// Mitsubishi GX Works2 project: 0206 MPS회로   PLC: Q03UDV

PROGRAM MAIN
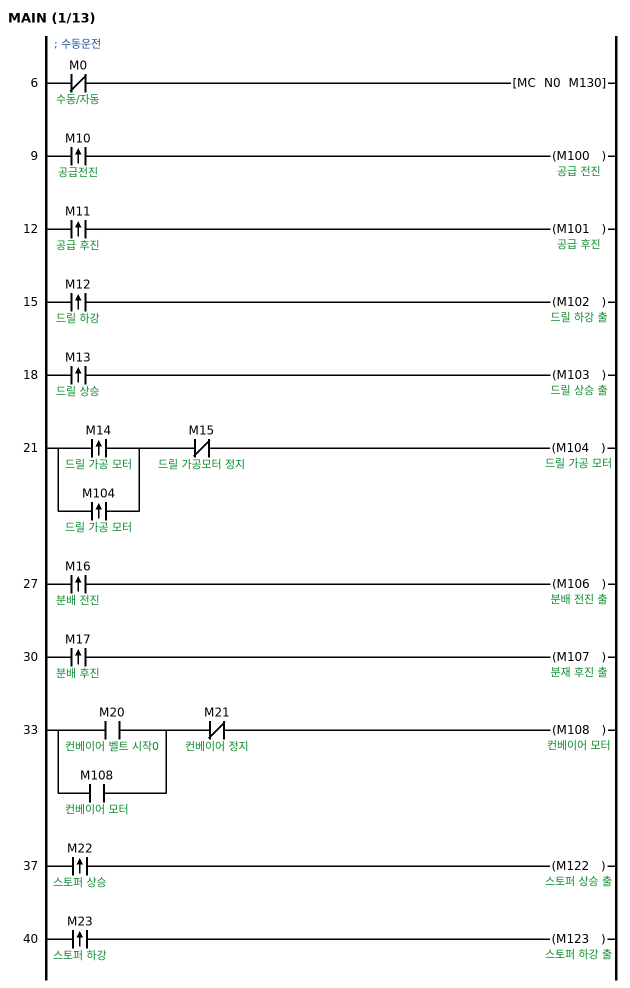
; 수동운전
6     LDI     M0  ; 수동/자동
      MC      N0 M130
9     LDP     M10  ; 공급전진
      OUT     M100  ; 공급 전진
12    LDP     M11  ; 공급 후진
      OUT     M101  ; 공급 후진
15    LDP     M12  ; 드릴 하강
      OUT     M102  ; 드릴 하강 출
18    LDP     M13  ; 드릴 상승
      OUT     M103  ; 드릴 상승 출
21    LDP     M14  ; 드릴 가공 모터
      ORP     M104  ; 드릴 가공 모터
      ANI     M15  ; 드릴 가공모터 정지
      OUT     M104  ; 드릴 가공 모터
27    LDP     M16  ; 분배 전진
      OUT     M106  ; 분배 전진 출
30    LDP     M17  ; 분배 후진
      OUT     M107  ; 분재 후진 출
33    LD      M20  ; 컨베이어 벨트 시작0
      OR      M108  ; 컨베이어 모터
      ANI     M21  ; 컨베이어 정지
      OUT     M108  ; 컨베이어 모터
37    LDP     M22  ; 스토퍼 상승
      OUT     M122  ; 스토퍼 상승 출
40    LDP     M23  ; 스토퍼 하강
      OUT     M123  ; 스토퍼 하강 출
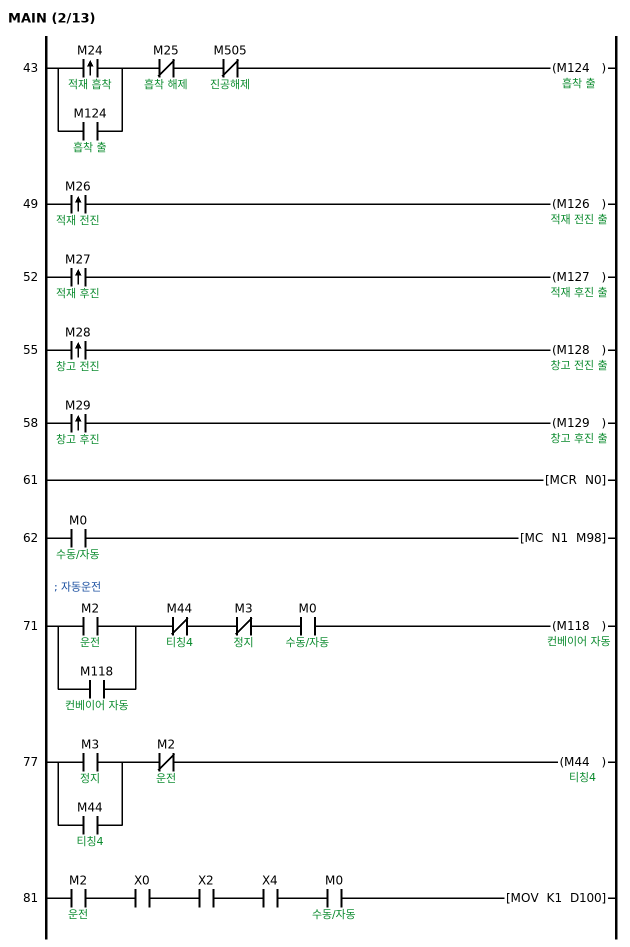
43    LDP     M24  ; 적재 흡착
      OR      M124  ; 흡착 출
      ANI     M25  ; 흡착 해제
      ANI     M505  ; 진공해제
      OUT     M124  ; 흡착 출
49    LDP     M26  ; 적재 전진
      OUT     M126  ; 적재 전진 출
52    LDP     M27  ; 적재 후진
      OUT     M127  ; 적재 후진 출
55    LDP     M28  ; 창고 전진
      OUT     M128  ; 창고 전진 출
58    LDP     M29  ; 창고 후진
      OUT     M129  ; 창고 후진 출
61    MCR     N0
62    LD      M0  ; 수동/자동
      MC      N1 M98
; 자동운전
71    LD      M2  ; 운전
      OR      M118  ; 컨베이어 자동
      ANI     M44  ; 티칭4
      ANI     M3  ; 정지
      AND     M0  ; 수동/자동
      OUT     M118  ; 컨베이어 자동
77    LD      M3  ; 정지
      OR      M44  ; 티칭4
      ANI     M2  ; 운전
      OUT     M44  ; 티칭4
81    LD      M2  ; 운전
      AND     X0
      AND     X2
      AND     X4
      AND     M0  ; 수동/자동
      MOV     K1 D100
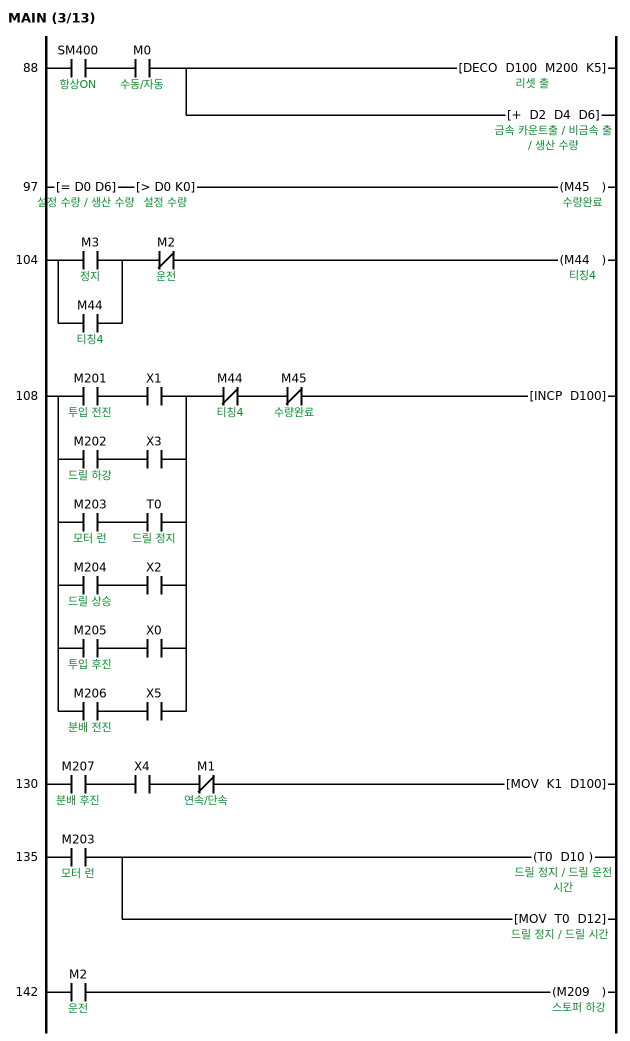
88    LD      SM400  ; 항상ON
      AND     M0  ; 수동/자동
      DECO    D100 M200 K5  ; 리셋 출
      +       D2 D4 D6  ; 금속 카운트출 / 비금속 출 / 생산 수량
97    LD=     D0 D6  ; 설정 수량 / 생산 수량
      AND>    D0 K0  ; 설정 수량
      OUT     M45  ; 수량완료
104   LD      M3  ; 정지
      OR      M44  ; 티칭4
      ANI     M2  ; 운전
      OUT     M44  ; 티칭4
108   LD      M201  ; 투입 전진
      AND     X1
      LD      M202  ; 드릴 하강
      AND     X3
      ORB
      LD      M203  ; 모터 런
      AND     T0  ; 드릴 정지
      ORB
      LD      M204  ; 드릴 상승
      AND     X2
      ORB
      LD      M205  ; 투입 후진
      AND     X0
      ORB
      LD      M206  ; 분배 전진
      AND     X5
      ORB
      ANI     M44  ; 티칭4
      ANI     M45  ; 수량완료
      INCP    D100
130   LD      M207  ; 분배 후진
      AND     X4
      ANI     M1  ; 연속/단속
      MOV     K1 D100
135   LD      M203  ; 모터 런
      OUT     T0 D10  ; 드릴 정지 / 드릴 운전 시간
      MOV     T0 D12  ; 드릴 시간
142   LD      M2  ; 운전
      OUT     M209  ; 스토퍼 하강
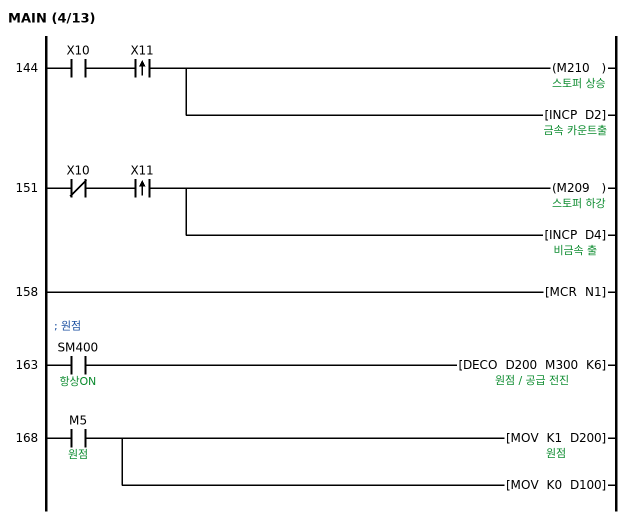
144   LD      X10
      ANDP    X11
      OUT     M210  ; 스토퍼 상승
      INCP    D2
151   LDI     X10
      ANDP    X11
      OUT     M209  ; 스토퍼 하강
      INCP    D4
158   MCR     N1
; 원점
163   LD      SM400  ; 항상ON
      DECO    D200 M300 K6  ; 원점 / 공급 전진
168   LD      M5  ; 원점
      MOV     K1 D200
      MOV     K0 D100
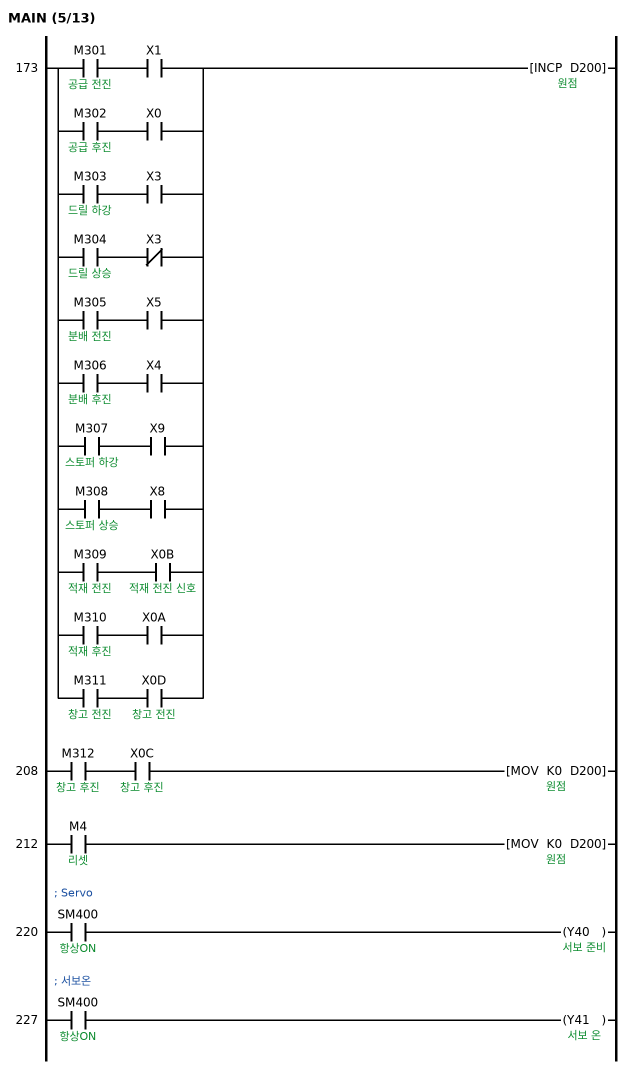
173   LD      M301  ; 공급 전진
      AND     X1
      LD      M302  ; 공급 후진
      AND     X0
      ORB
      LD      M303  ; 드릴 하강
      AND     X3
      ORB
      LD      M304  ; 드릴 상승
      ANI     X3
      ORB
      LD      M305  ; 분배 전진
      AND     X5
      ORB
      LD      M306  ; 분배 후진
      AND     X4
      ORB
      LD      M307  ; 스토퍼 하강
      AND     X9
      ORB
      LD      M308  ; 스토퍼 상승
      AND     X8
      ORB
      LD      M309  ; 적재 전진
      AND     X0B  ; 적재 전진 신호
      ORB
      LD      M310  ; 적재 후진
      AND     X0A
      ORB
      LD      M311  ; 창고 전진
      AND     X0D  ; 창고 전진
      ORB
      INCP    D200
208   LD      M312  ; 창고 후진
      AND     X0C  ; 창고 후진
      MOV     K0 D200
212   LD      M4  ; 리셋
      MOV     K0 D200
; Servo
220   LD      SM400  ; 항상ON
      OUT     Y40  ; 서보 준비
; 서보온
227   LD      SM400  ; 항상ON
      OUT     Y41  ; 서보 온
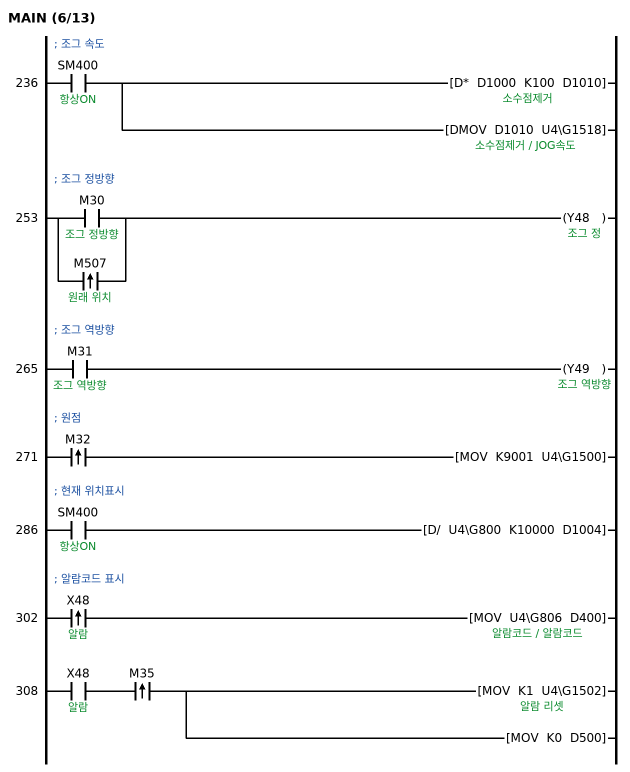
; 조그 속도
236   LD      SM400  ; 항상ON
      D*      D1000 K100 D1010  ; 소수점제거
      DMOV    D1010 U4\G1518  ; JOG속도
; 조그 정방향
253   LD      M30  ; 조그 정방향
      ORP     M507  ; 원래 위치
      OUT     Y48  ; 조그 정
; 조그 역방향
265   LD      M31  ; 조그 역방향
      OUT     Y49  ; 조그 역방향
; 원점
271   LDP     M32
      MOV     K9001 U4\G1500
; 현재 위치표시
286   LD      SM400  ; 항상ON
      D/      U4\G800 K10000 D1004
; 알람코드 표시
302   LDP     X48  ; 알람
      MOV     U4\G806 D400  ; 알람코드 / 알람코드
308   LD      X48  ; 알람
      ANDP    M35
      MOV     K1 U4\G1502  ; 알람 리셋
      MOV     K0 D500
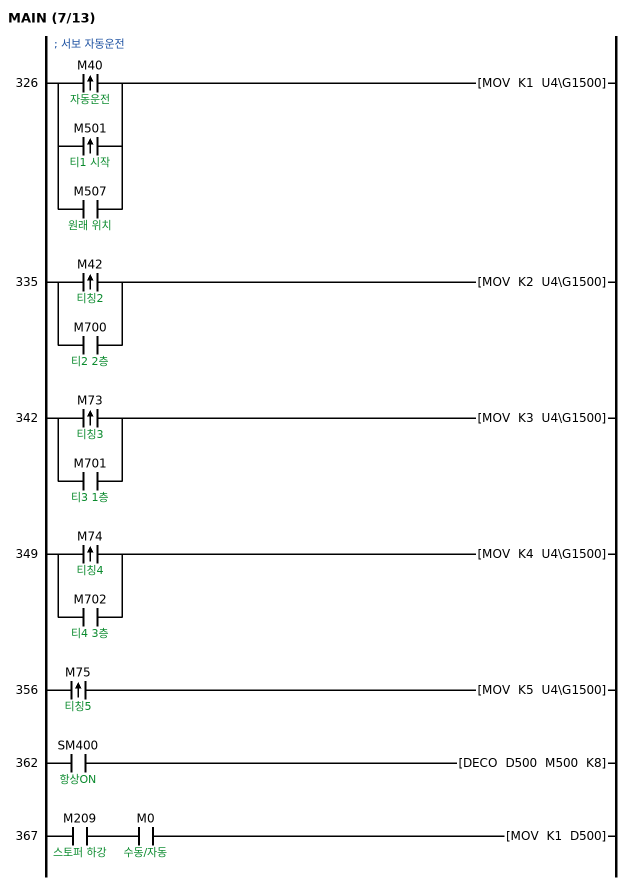
; 서보 자동운전
326   LDP     M40  ; 자동운전
      ORP     M501  ; 티1 시작
      OR      M507  ; 원래 위치
      MOV     K1 U4\G1500
335   LDP     M42  ; 티칭2
      OR      M700  ; 티2 2층
      MOV     K2 U4\G1500
342   LDP     M73  ; 티칭3
      OR      M701  ; 티3 1층
      MOV     K3 U4\G1500
349   LDP     M74  ; 티칭4
      OR      M702  ; 티4 3층
      MOV     K4 U4\G1500
356   LDP     M75  ; 티칭5
      MOV     K5 U4\G1500
362   LD      SM400  ; 항상ON
      DECO    D500 M500 K8
367   LD      M209  ; 스토퍼 하강
      AND     M0  ; 수동/자동
      MOV     K1 D500
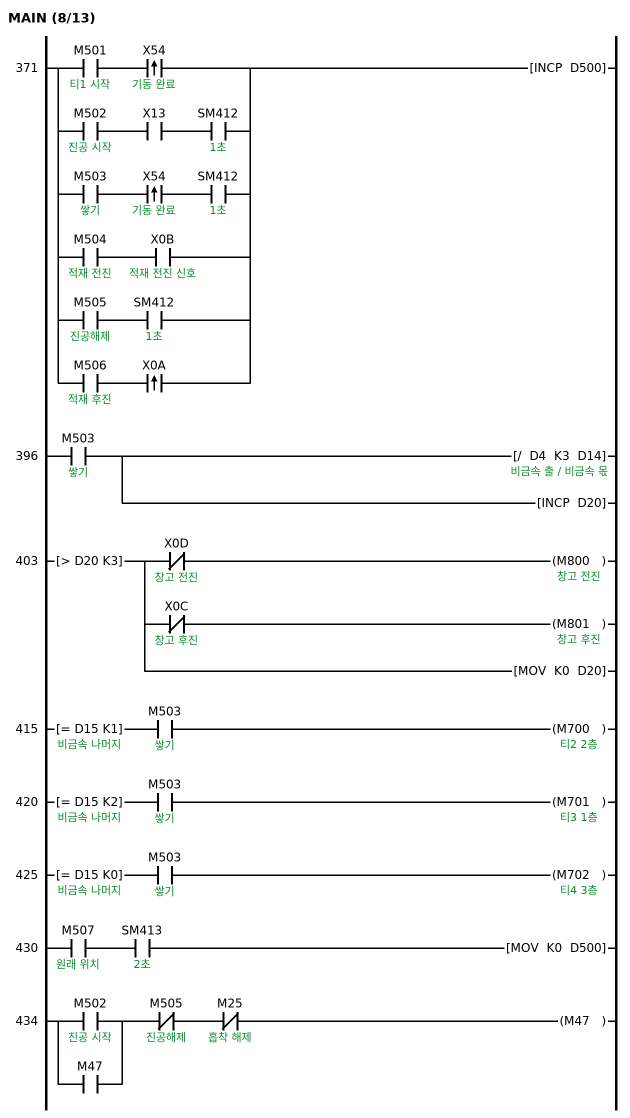
371   LD      M501  ; 티1 시작
      ANDP    X54  ; 기동 완료
      LD      M502  ; 진공 시작
      AND     X13
      AND     SM412  ; 1초
      ORB
      LD      M503  ; 쌓기
      ANDP    X54  ; 기동 완료
      AND     SM412  ; 1초
      ORB
      LD      M504  ; 적재 전진
      AND     X0B  ; 적재 전진 신호
      ORB
      LD      M505  ; 진공해제
      AND     SM412  ; 1초
      ORB
      LD      M506  ; 적재 후진
      ANDP    X0A
      ORB
      INCP    D500
396   LD      M503  ; 쌓기
      /       D4 K3 D14  ; 비금속 몫
      INCP    D20
403   LD>     D20 K3
      MPS
      ANI     X0D  ; 창고 전진
      OUT     M800  ; 창고 전진
      MRD
      ANI     X0C  ; 창고 후진
      OUT     M801  ; 창고 후진
      MPP
      MOV     K0 D20
415   LD=     D15 K1  ; 비금속 나머지
      AND     M503  ; 쌓기
      OUT     M700  ; 티2 2층
420   LD=     D15 K2  ; 비금속 나머지
      AND     M503  ; 쌓기
      OUT     M701  ; 티3 1층
425   LD=     D15 K0  ; 비금속 나머지
      AND     M503  ; 쌓기
      OUT     M702  ; 티4 3층
430   LD      M507  ; 원래 위치
      AND     SM413  ; 2초
      MOV     K0 D500
434   LD      M502  ; 진공 시작
      OR      M47
      ANI     M505  ; 진공해제
      ANI     M25  ; 흡착 해제
      OUT     M47
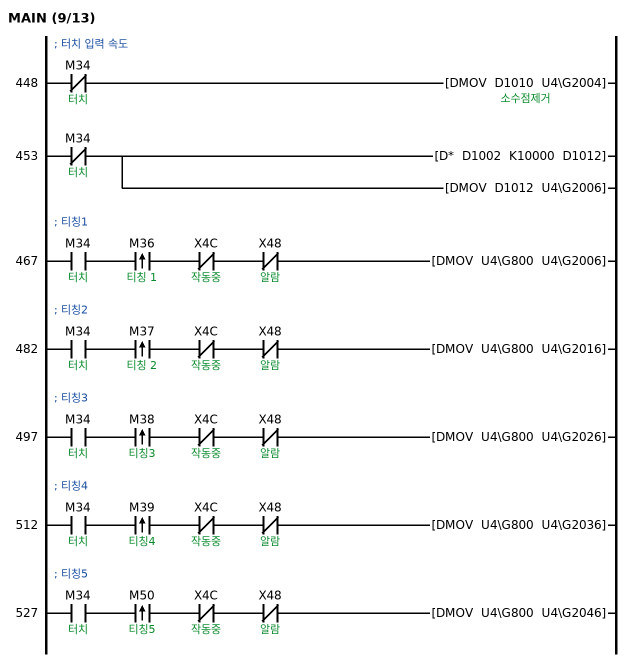
; 터치 입력 속도
448   LDI     M34  ; 터치
      DMOV    D1010 U4\G2004
453   LDI     M34  ; 터치
      D*      D1002 K10000 D1012
      DMOV    D1012 U4\G2006
; 티칭1
467   LD      M34  ; 터치
      ANDP    M36  ; 티칭 1
      ANI     X4C  ; 작동중
      ANI     X48  ; 알람
      DMOV    U4\G800 U4\G2006
; 티칭2
482   LD      M34  ; 터치
      ANDP    M37  ; 티칭 2
      ANI     X4C  ; 작동중
      ANI     X48  ; 알람
      DMOV    U4\G800 U4\G2016
; 티칭3
497   LD      M34  ; 터치
      ANDP    M38  ; 티칭3
      ANI     X4C  ; 작동중
      ANI     X48  ; 알람
      DMOV    U4\G800 U4\G2026
; 티칭4
512   LD      M34  ; 터치
      ANDP    M39  ; 티칭4
      ANI     X4C  ; 작동중
      ANI     X48  ; 알람
      DMOV    U4\G800 U4\G2036
; 티칭5
527   LD      M34  ; 터치
      ANDP    M50  ; 티칭5
      ANI     X4C  ; 작동중
      ANI     X48  ; 알람
      DMOV    U4\G800 U4\G2046
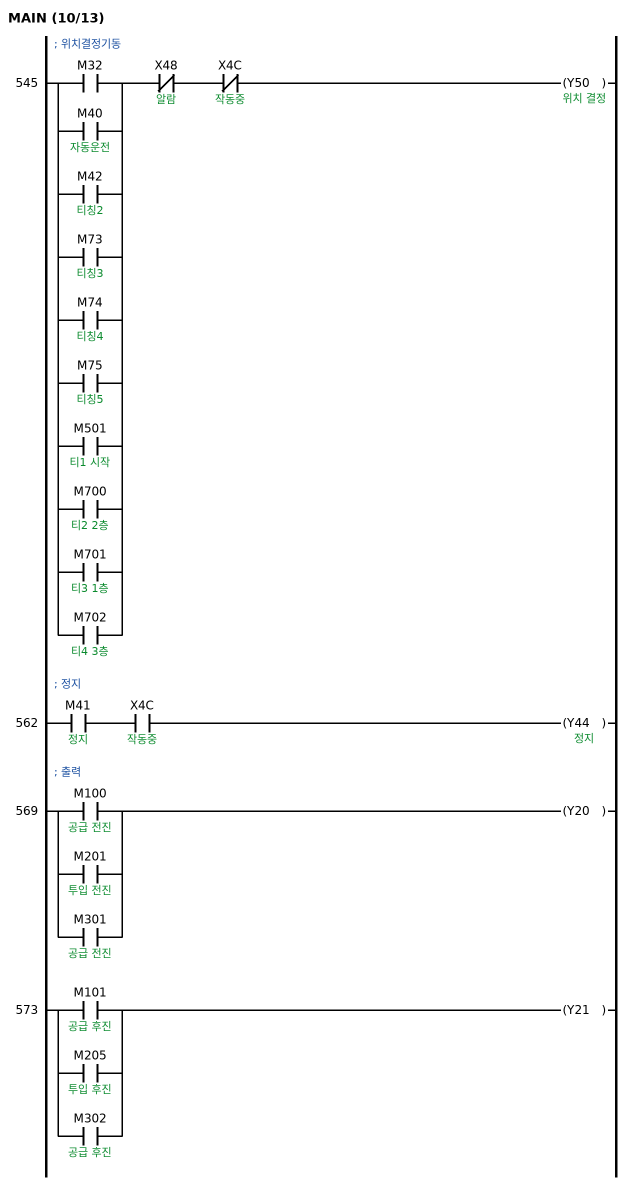
; 위치결정기동
545   LD      M32
      OR      M40  ; 자동운전
      OR      M42  ; 티칭2
      OR      M73  ; 티칭3
      OR      M74  ; 티칭4
      OR      M75  ; 티칭5
      OR      M501  ; 티1 시작
      OR      M700  ; 티2 2층
      OR      M701  ; 티3 1층
      OR      M702  ; 티4 3층
      ANI     X48  ; 알람
      ANI     X4C  ; 작동중
      OUT     Y50  ; 위치 결정
; 정지
562   LD      M41  ; 정지
      AND     X4C  ; 작동중
      OUT     Y44  ; 정지
; 출력
569   LD      M100  ; 공급 전진
      OR      M201  ; 투입 전진
      OR      M301  ; 공급 전진
      OUT     Y20
573   LD      M101  ; 공급 후진
      OR      M205  ; 투입 후진
      OR      M302  ; 공급 후진
      OUT     Y21
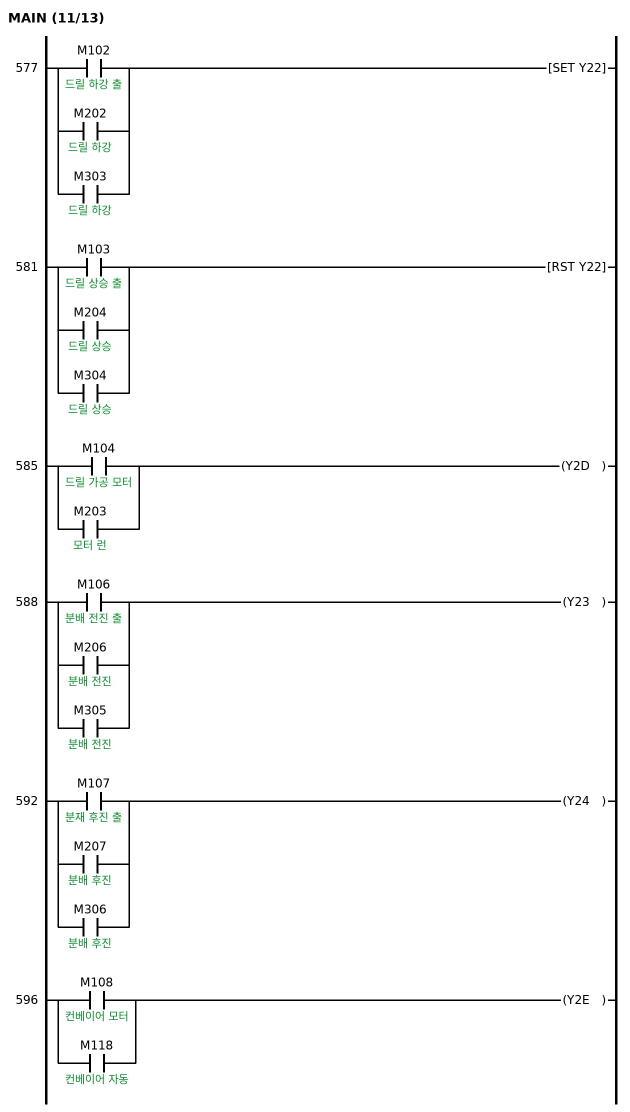
577   LD      M102  ; 드릴 하강 출
      OR      M202  ; 드릴 하강
      OR      M303  ; 드릴 하강
      SET     Y22
581   LD      M103  ; 드릴 상승 출
      OR      M204  ; 드릴 상승
      OR      M304  ; 드릴 상승
      RST     Y22
585   LD      M104  ; 드릴 가공 모터
      OR      M203  ; 모터 런
      OUT     Y2D
588   LD      M106  ; 분배 전진 출
      OR      M206  ; 분배 전진
      OR      M305  ; 분배 전진
      OUT     Y23
592   LD      M107  ; 분재 후진 출
      OR      M207  ; 분배 후진
      OR      M306  ; 분배 후진
      OUT     Y24
596   LD      M108  ; 컨베이어 모터
      OR      M118  ; 컨베이어 자동
      OUT     Y2E
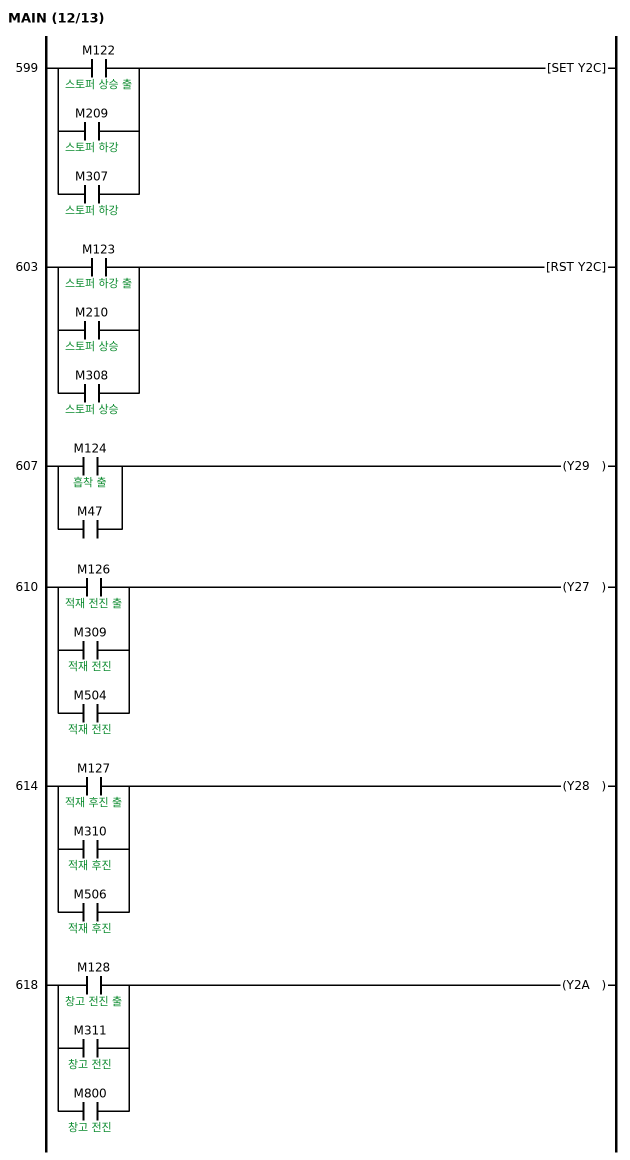
599   LD      M122  ; 스토퍼 상승 출
      OR      M209  ; 스토퍼 하강
      OR      M307  ; 스토퍼 하강
      SET     Y2C
603   LD      M123  ; 스토퍼 하강 출
      OR      M210  ; 스토퍼 상승
      OR      M308  ; 스토퍼 상승
      RST     Y2C
607   LD      M124  ; 흡착 출
      OR      M47
      OUT     Y29
610   LD      M126  ; 적재 전진 출
      OR      M309  ; 적재 전진
      OR      M504  ; 적재 전진
      OUT     Y27
614   LD      M127  ; 적재 후진 출
      OR      M310  ; 적재 후진
      OR      M506  ; 적재 후진
      OUT     Y28
618   LD      M128  ; 창고 전진 출
      OR      M311  ; 창고 전진
      OR      M800  ; 창고 전진
      OUT     Y2A
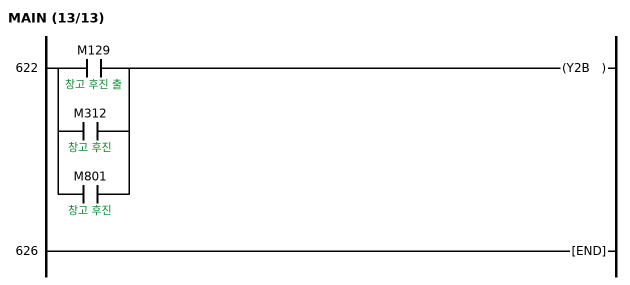
622   LD      M129  ; 창고 후진 출
      OR      M312  ; 창고 후진
      OR      M801  ; 창고 후진
      OUT     Y2B
626   END
END_PROGRAM

// device comments not shown above
M43  ; 티칭3
M54  ; 티칭 4
M55  ; 티칭5
M105  ; 분배 전진 출
M150  ; 원점릴레링
M508  ; 티1 시작
M509  ; 진공 시작
M510  ; 티3 시작
M511  ; 적재 진진
M512  ; 진공 해제
M513  ; 적재 후진
M514  ; 원래 위치
M515  ; 티1 시작
M516  ; 진공 시작
M517  ; 티4 시작
M518  ; 적재 직진
M519  ; 진공 해제
M520  ; 적재 후진
M521  ; 원래 위치
M522  ; 창고 위치
M600  ; 비금속 검출
X12  ; 스토퍼 검출
X50  ; 기동 완료
X204  ; 투입 후진
X304  ; 드릴 상승
X305  ; 분배 전진
X406  ; 분배 후진
C0  ; 금속 카운트
C1  ; 비금속
C2  ; 생산수량
